{attribute addProperty BoxType "EL2521-0000-1019"}
{attribute addProperty Id "Sel_Ack_End_counterBIT10.1251Ramp_activeBIT10.1252Status_of_input_targetBIT10.1255Status_of_input_zeroBIT10.1256ErrorBIT10.1257Sync_errorBIT10.12532TxPDO_ToggleBIT10.1259"}
{attribute addProperty CRC "3534717475"}
{attribute addProperty SizeInBites "16"}
{attribute addProperty SizeInBytes "2"}
TYPE Status_D2AF8223 :
STRUCT
	{attribute addProperty Name "Sel_Ack_End_counter"}
	Sel_Ack_End_counter : BIT;
	{attribute addProperty Name "Ramp_active"}
	Ramp_active : BIT;
	{attribute 'hide'}
	reserve_1_BIT_0 : BIT;
	{attribute 'hide'}
	reserve_1_BIT_1 : BIT;
	{attribute addProperty Name "Status_of_input_target"}
	Status_of_input_target : BIT;
	{attribute addProperty Name "Status_of_input_zero"}
	Status_of_input_zero : BIT;
	{attribute addProperty Name "Error"}
	Error : BIT;
	{attribute 'hide'}
	reserve_2_BIT_0 : BIT;
	{attribute 'hide'}
	reserve_2_BIT_1 : BIT;
	{attribute 'hide'}
	reserve_2_BIT_2 : BIT;
	{attribute 'hide'}
	reserve_2_BIT_3 : BIT;
	{attribute 'hide'}
	reserve_2_BIT_4 : BIT;
	{attribute 'hide'}
	reserve_2_BIT_5 : BIT;
	{attribute addProperty Name "Sync_error"}
	Sync_error : BIT;
	{attribute 'hide'}
	reserve_3 : BIT;
	{attribute addProperty Name "TxPDO_Toggle"}
	TxPDO_Toggle : BIT;
END_STRUCT
END_TYPE

(* stored: Version 1.2.0.0, ProductVersion 3.1.4024.9
   DUT Status_D2AF8223: Id {d074dd5c-28e1-433f-b1d8-70c9f2c7ad0d} *)
